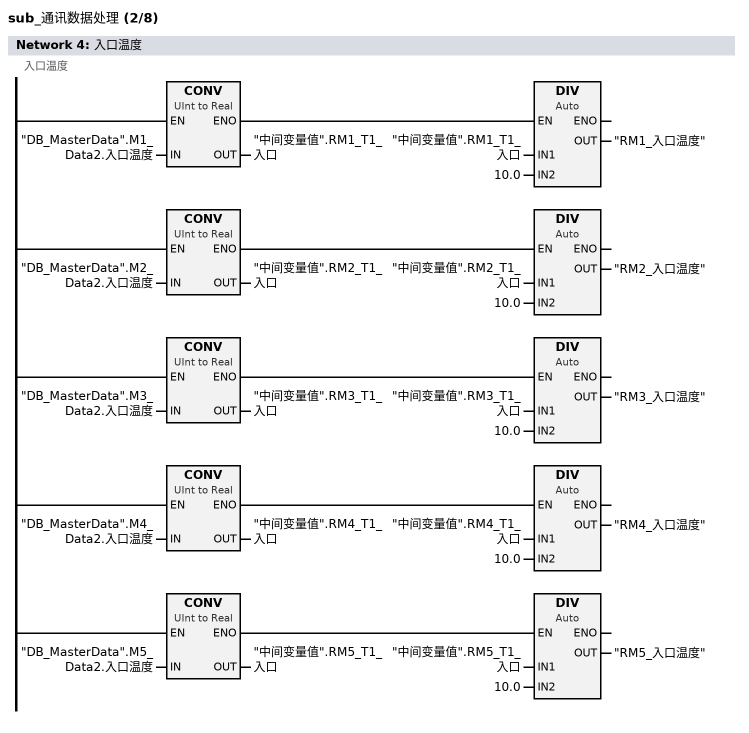
   RUNG wire#powerrail
      { S7_Templates := "[SrcType := UInt, DestType := Real]" } Convert(in := "DB_MasterData".M1_Data2.入口温度, out => "中间变量值".RM1_T1_入口)
      Div(in1 := "中间变量值".RM1_T1_入口, in2 := 10.0, out => "RM1_入口温度")
   END_RUNG
   RUNG wire#powerrail
      { S7_Templates := "[SrcType := UInt, DestType := Real]" } Convert(in := "DB_MasterData".M2_Data2.入口温度, out => "中间变量值".RM2_T1_入口)
      Div(in1 := "中间变量值".RM2_T1_入口, in2 := 10.0, out => "RM2_入口温度")
   END_RUNG
   RUNG wire#powerrail
      { S7_Templates := "[SrcType := UInt, DestType := Real]" } Convert(in := "DB_MasterData".M3_Data2.入口温度, out => "中间变量值".RM3_T1_入口)
      Div(in1 := "中间变量值".RM3_T1_入口, in2 := 10.0, out => "RM3_入口温度")
   END_RUNG
   RUNG wire#powerrail
      { S7_Templates := "[SrcType := UInt, DestType := Real]" } Convert(in := "DB_MasterData".M4_Data2.入口温度, out => "中间变量值".RM4_T1_入口)
      Div(in1 := "中间变量值".RM4_T1_入口, in2 := 10.0, out => "RM4_入口温度")
   END_RUNG
   RUNG wire#powerrail
      { S7_Templates := "[SrcType := UInt, DestType := Real]" } Convert(in := "DB_MasterData".M5_Data2.入口温度, out => "中间变量值".RM5_T1_入口)
      Div(in1 := "中间变量值".RM5_T1_入口, in2 := 10.0, out => "RM5_入口温度")
   END_RUNG
   // the same network as SCL:
   "中间变量值".RM1_T1_入口 := UINT_TO_REAL("DB_MasterData".M1_Data2.入口温度);
   "RM1_入口温度" := "中间变量值".RM1_T1_入口 / 10.0;
   "中间变量值".RM2_T1_入口 := UINT_TO_REAL("DB_MasterData".M2_Data2.入口温度);
   "RM2_入口温度" := "中间变量值".RM2_T1_入口 / 10.0;
   "中间变量值".RM3_T1_入口 := UINT_TO_REAL("DB_MasterData".M3_Data2.入口温度);
   "RM3_入口温度" := "中间变量值".RM3_T1_入口 / 10.0;
   "中间变量值".RM4_T1_入口 := UINT_TO_REAL("DB_MasterData".M4_Data2.入口温度);
   "RM4_入口温度" := "中间变量值".RM4_T1_入口 / 10.0;
   "中间变量值".RM5_T1_入口 := UINT_TO_REAL("DB_MasterData".M5_Data2.入口温度);
   "RM5_入口温度" := "中间变量值".RM5_T1_入口 / 10.0;
END_REGION

REGION Network 5: 出口温度
   // 出口温度
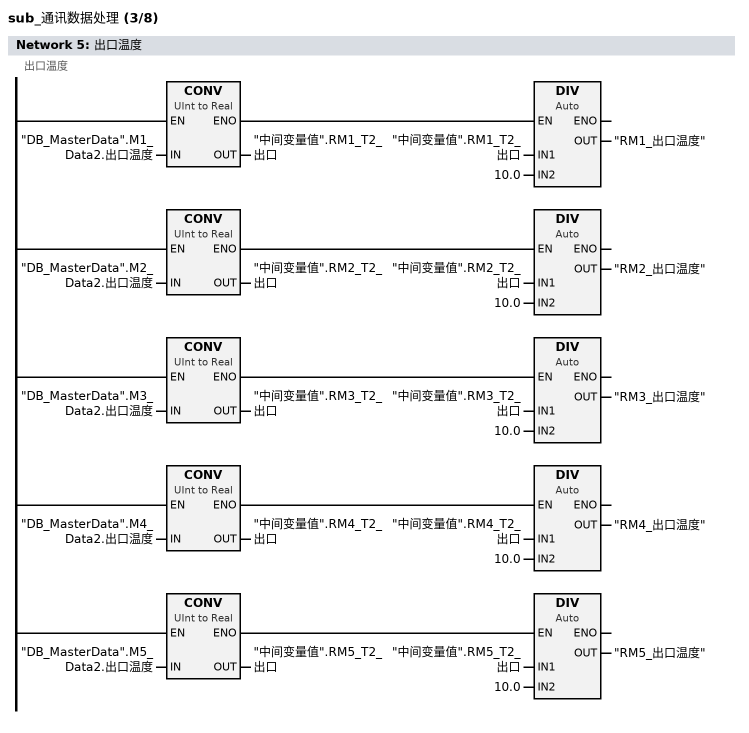
   RUNG wire#powerrail
      { S7_Templates := "[SrcType := UInt, DestType := Real]" } Convert(in := "DB_MasterData".M1_Data2.出口温度, out => "中间变量值".RM1_T2_出口)
      Div(in1 := "中间变量值".RM1_T2_出口, in2 := 10.0, out => "RM1_出口温度")
   END_RUNG
   RUNG wire#powerrail
      { S7_Templates := "[SrcType := UInt, DestType := Real]" } Convert(in := "DB_MasterData".M2_Data2.出口温度, out => "中间变量值".RM2_T2_出口)
      Div(in1 := "中间变量值".RM2_T2_出口, in2 := 10.0, out => "RM2_出口温度")
   END_RUNG
   RUNG wire#powerrail
      { S7_Templates := "[SrcType := UInt, DestType := Real]" } Convert(in := "DB_MasterData".M3_Data2.出口温度, out => "中间变量值".RM3_T2_出口)
      Div(in1 := "中间变量值".RM3_T2_出口, in2 := 10.0, out => "RM3_出口温度")
   END_RUNG
   RUNG wire#powerrail
      { S7_Templates := "[SrcType := UInt, DestType := Real]" } Convert(in := "DB_MasterData".M4_Data2.出口温度, out => "中间变量值".RM4_T2_出口)
      Div(in1 := "中间变量值".RM4_T2_出口, in2 := 10.0, out => "RM4_出口温度")
   END_RUNG
   RUNG wire#powerrail
      { S7_Templates := "[SrcType := UInt, DestType := Real]" } Convert(in := "DB_MasterData".M5_Data2.出口温度, out => "中间变量值".RM5_T2_出口)
      Div(in1 := "中间变量值".RM5_T2_出口, in2 := 10.0, out => "RM5_出口温度")
   END_RUNG
   // the same network as SCL:
   "中间变量值".RM1_T2_出口 := UINT_TO_REAL("DB_MasterData".M1_Data2.出口温度);
   "RM1_出口温度" := "中间变量值".RM1_T2_出口 / 10.0;
   "中间变量值".RM2_T2_出口 := UINT_TO_REAL("DB_MasterData".M2_Data2.出口温度);
   "RM2_出口温度" := "中间变量值".RM2_T2_出口 / 10.0;
   "中间变量值".RM3_T2_出口 := UINT_TO_REAL("DB_MasterData".M3_Data2.出口温度);
   "RM3_出口温度" := "中间变量值".RM3_T2_出口 / 10.0;
   "中间变量值".RM4_T2_出口 := UINT_TO_REAL("DB_MasterData".M4_Data2.出口温度);
   "RM4_出口温度" := "中间变量值".RM4_T2_出口 / 10.0;
   "中间变量值".RM5_T2_出口 := UINT_TO_REAL("DB_MasterData".M5_Data2.出口温度);
   "RM5_出口温度" := "中间变量值".RM5_T2_出口 / 10.0;
END_REGION

REGION Network 7: #1 吸收式热泵数据-温度
   // #1 吸收式热泵数据
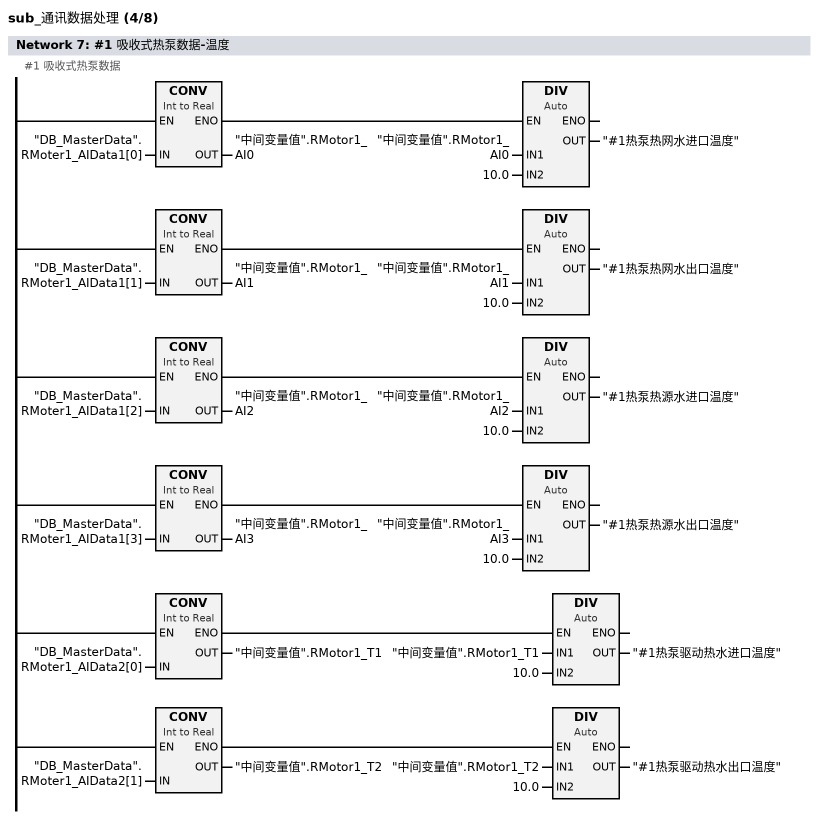
   RUNG wire#powerrail
      { S7_Templates := "[SrcType := Int, DestType := Real]" } Convert(in := "DB_MasterData".RMoter1_AIData1[0], out => "中间变量值".RMotor1_AI0)
      Div(in1 := "中间变量值".RMotor1_AI0, in2 := 10.0, out => "#1热泵热网水进口温度")
   END_RUNG
   RUNG wire#powerrail
      { S7_Templates := "[SrcType := Int, DestType := Real]" } Convert(in := "DB_MasterData".RMoter1_AIData1[1], out => "中间变量值".RMotor1_AI1)
      Div(in1 := "中间变量值".RMotor1_AI1, in2 := 10.0, out => "#1热泵热网水出口温度")
   END_RUNG
   RUNG wire#powerrail
      { S7_Templates := "[SrcType := Int, DestType := Real]" } Convert(in := "DB_MasterData".RMoter1_AIData1[2], out => "中间变量值".RMotor1_AI2)
      Div(in1 := "中间变量值".RMotor1_AI2, in2 := 10.0, out => "#1热泵热源水进口温度")
   END_RUNG
   RUNG wire#powerrail
      { S7_Templates := "[SrcType := Int, DestType := Real]" } Convert(in := "DB_MasterData".RMoter1_AIData1[3], out => "中间变量值".RMotor1_AI3)
      Div(in1 := "中间变量值".RMotor1_AI3, in2 := 10.0, out => "#1热泵热源水出口温度")
   END_RUNG
   RUNG wire#powerrail
      { S7_Templates := "[SrcType := Int, DestType := Real]" } Convert(in := "DB_MasterData".RMoter1_AIData2[0], out => "中间变量值".RMotor1_T1)
      Div(in1 := "中间变量值".RMotor1_T1, in2 := 10.0, out => "#1热泵驱动热水进口温度")
   END_RUNG
   RUNG wire#powerrail
      { S7_Templates := "[SrcType := Int, DestType := Real]" } Convert(in := "DB_MasterData".RMoter1_AIData2[1], out => "中间变量值".RMotor1_T2)
      Div(in1 := "中间变量值".RMotor1_T2, in2 := 10.0, out => "#1热泵驱动热水出口温度")
   END_RUNG
   // the same network as SCL:
   "中间变量值".RMotor1_AI0 := INT_TO_REAL("DB_MasterData".RMoter1_AIData1[0]);
   "#1热泵热网水进口温度" := "中间变量值".RMotor1_AI0 / 10.0;
   "中间变量值".RMotor1_AI1 := INT_TO_REAL("DB_MasterData".RMoter1_AIData1[1]);
   "#1热泵热网水出口温度" := "中间变量值".RMotor1_AI1 / 10.0;
   "中间变量值".RMotor1_AI2 := INT_TO_REAL("DB_MasterData".RMoter1_AIData1[2]);
   "#1热泵热源水进口温度" := "中间变量值".RMotor1_AI2 / 10.0;
   "中间变量值".RMotor1_AI3 := INT_TO_REAL("DB_MasterData".RMoter1_AIData1[3]);
   "#1热泵热源水出口温度" := "中间变量值".RMotor1_AI3 / 10.0;
   "中间变量值".RMotor1_T1 := INT_TO_REAL("DB_MasterData".RMoter1_AIData2[0]);
   "#1热泵驱动热水进口温度" := "中间变量值".RMotor1_T1 / 10.0;
   "中间变量值".RMotor1_T2 := INT_TO_REAL("DB_MasterData".RMoter1_AIData2[1]);
   "#1热泵驱动热水出口温度" := "中间变量值".RMotor1_T2 / 10.0;
END_REGION

REGION Network 8: #1 吸收式热泵数据-压力
   // #1 吸收式热泵数据-压力
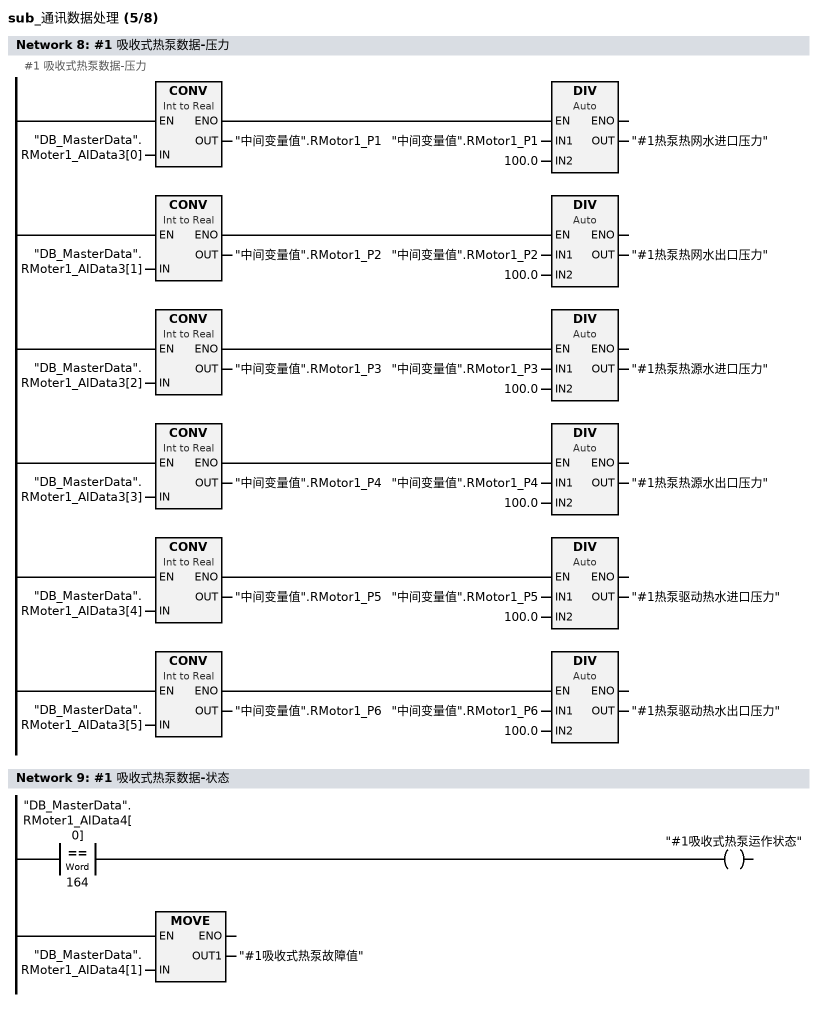
   RUNG wire#powerrail
      { S7_Templates := "[SrcType := Int, DestType := Real]" } Convert(in := "DB_MasterData".RMoter1_AIData3[0], out => "中间变量值".RMotor1_P1)
      Div(in1 := "中间变量值".RMotor1_P1, in2 := 100.0, out => "#1热泵热网水进口压力")
   END_RUNG
   RUNG wire#powerrail
      { S7_Templates := "[SrcType := Int, DestType := Real]" } Convert(in := "DB_MasterData".RMoter1_AIData3[1], out => "中间变量值".RMotor1_P2)
      Div(in1 := "中间变量值".RMotor1_P2, in2 := 100.0, out => "#1热泵热网水出口压力")
   END_RUNG
   RUNG wire#powerrail
      { S7_Templates := "[SrcType := Int, DestType := Real]" } Convert(in := "DB_MasterData".RMoter1_AIData3[2], out => "中间变量值".RMotor1_P3)
      Div(in1 := "中间变量值".RMotor1_P3, in2 := 100.0, out => "#1热泵热源水进口压力")
   END_RUNG
   RUNG wire#powerrail
      { S7_Templates := "[SrcType := Int, DestType := Real]" } Convert(in := "DB_MasterData".RMoter1_AIData3[3], out => "中间变量值".RMotor1_P4)
      Div(in1 := "中间变量值".RMotor1_P4, in2 := 100.0, out => "#1热泵热源水出口压力")
   END_RUNG
   RUNG wire#powerrail
      { S7_Templates := "[SrcType := Int, DestType := Real]" } Convert(in := "DB_MasterData".RMoter1_AIData3[4], out => "中间变量值".RMotor1_P5)
      Div(in1 := "中间变量值".RMotor1_P5, in2 := 100.0, out => "#1热泵驱动热水进口压力")
   END_RUNG
   RUNG wire#powerrail
      { S7_Templates := "[SrcType := Int, DestType := Real]" } Convert(in := "DB_MasterData".RMoter1_AIData3[5], out => "中间变量值".RMotor1_P6)
      Div(in1 := "中间变量值".RMotor1_P6, in2 := 100.0, out => "#1热泵驱动热水出口压力")
   END_RUNG
   // the same network as SCL:
   "中间变量值".RMotor1_P1 := INT_TO_REAL("DB_MasterData".RMoter1_AIData3[0]);
   "#1热泵热网水进口压力" := "中间变量值".RMotor1_P1 / 100.0;
   "中间变量值".RMotor1_P2 := INT_TO_REAL("DB_MasterData".RMoter1_AIData3[1]);
   "#1热泵热网水出口压力" := "中间变量值".RMotor1_P2 / 100.0;
   "中间变量值".RMotor1_P3 := INT_TO_REAL("DB_MasterData".RMoter1_AIData3[2]);
   "#1热泵热源水进口压力" := "中间变量值".RMotor1_P3 / 100.0;
   "中间变量值".RMotor1_P4 := INT_TO_REAL("DB_MasterData".RMoter1_AIData3[3]);
   "#1热泵热源水出口压力" := "中间变量值".RMotor1_P4 / 100.0;
   "中间变量值".RMotor1_P5 := INT_TO_REAL("DB_MasterData".RMoter1_AIData3[4]);
   "#1热泵驱动热水进口压力" := "中间变量值".RMotor1_P5 / 100.0;
   "中间变量值".RMotor1_P6 := INT_TO_REAL("DB_MasterData".RMoter1_AIData3[5]);
   "#1热泵驱动热水出口压力" := "中间变量值".RMotor1_P6 / 100.0;
END_REGION

REGION Network 9: #1 吸收式热泵数据-状态
   RUNG wire#powerrail
      { S7_Templates := "SrcType := Word" } EQ_Contact(in1 := "DB_MasterData".RMoter1_AIData4[0], in2 := 164)
      Coil( "#1吸收式热泵运作状态" )
   END_RUNG
   RUNG wire#powerrail
      Move(in := "DB_MasterData".RMoter1_AIData4[1], out1 => "#1吸收式热泵故障值")
   END_RUNG
   // the same network as SCL:
   "#1吸收式热泵运作状态" := "DB_MasterData".RMoter1_AIData4[0] = 164;
   "#1吸收式热泵故障值" := "DB_MasterData".RMoter1_AIData4[1];
END_REGION

REGION Network 10: #2 吸收式热泵数据-温度
   // #2 吸收式热泵数据
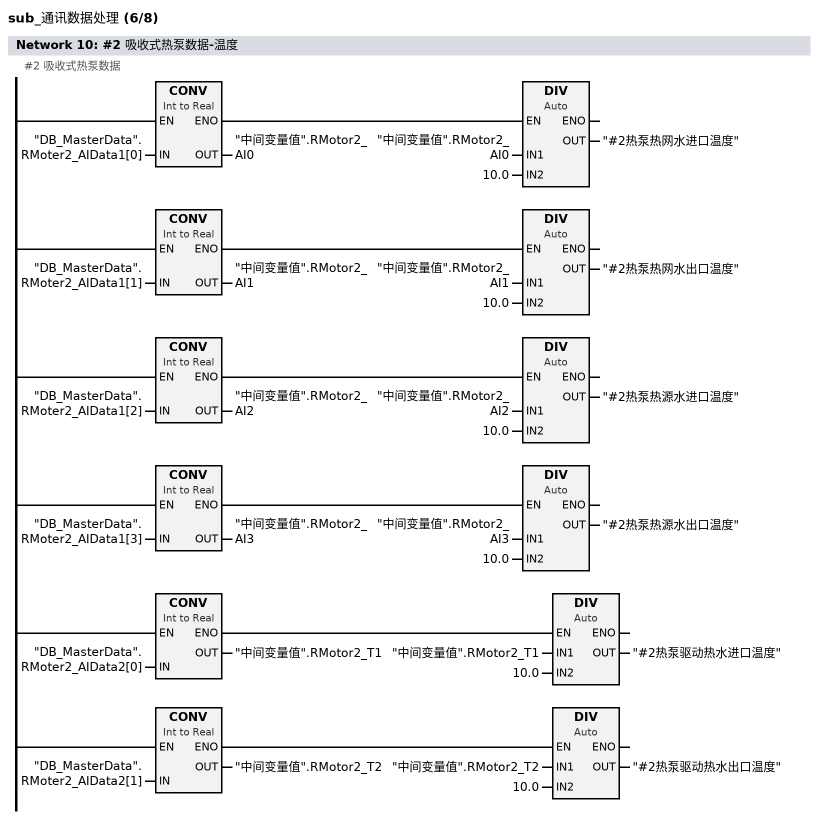
   RUNG wire#powerrail
      { S7_Templates := "[SrcType := Int, DestType := Real]" } Convert(in := "DB_MasterData".RMoter2_AIData1[0], out => "中间变量值".RMotor2_AI0)
      Div(in1 := "中间变量值".RMotor2_AI0, in2 := 10.0, out => "#2热泵热网水进口温度")
   END_RUNG
   RUNG wire#powerrail
      { S7_Templates := "[SrcType := Int, DestType := Real]" } Convert(in := "DB_MasterData".RMoter2_AIData1[1], out => "中间变量值".RMotor2_AI1)
      Div(in1 := "中间变量值".RMotor2_AI1, in2 := 10.0, out => "#2热泵热网水出口温度")
   END_RUNG
   RUNG wire#powerrail
      { S7_Templates := "[SrcType := Int, DestType := Real]" } Convert(in := "DB_MasterData".RMoter2_AIData1[2], out => "中间变量值".RMotor2_AI2)
      Div(in1 := "中间变量值".RMotor2_AI2, in2 := 10.0, out => "#2热泵热源水进口温度")
   END_RUNG
   RUNG wire#powerrail
      { S7_Templates := "[SrcType := Int, DestType := Real]" } Convert(in := "DB_MasterData".RMoter2_AIData1[3], out => "中间变量值".RMotor2_AI3)
      Div(in1 := "中间变量值".RMotor2_AI3, in2 := 10.0, out => "#2热泵热源水出口温度")
   END_RUNG
   RUNG wire#powerrail
      { S7_Templates := "[SrcType := Int, DestType := Real]" } Convert(in := "DB_MasterData".RMoter2_AIData2[0], out => "中间变量值".RMotor2_T1)
      Div(in1 := "中间变量值".RMotor2_T1, in2 := 10.0, out => "#2热泵驱动热水进口温度")
   END_RUNG
   RUNG wire#powerrail
      { S7_Templates := "[SrcType := Int, DestType := Real]" } Convert(in := "DB_MasterData".RMoter2_AIData2[1], out => "中间变量值".RMotor2_T2)
      Div(in1 := "中间变量值".RMotor2_T2, in2 := 10.0, out => "#2热泵驱动热水出口温度")
   END_RUNG
   // the same network as SCL:
   "中间变量值".RMotor2_AI0 := INT_TO_REAL("DB_MasterData".RMoter2_AIData1[0]);
   "#2热泵热网水进口温度" := "中间变量值".RMotor2_AI0 / 10.0;
   "中间变量值".RMotor2_AI1 := INT_TO_REAL("DB_MasterData".RMoter2_AIData1[1]);
   "#2热泵热网水出口温度" := "中间变量值".RMotor2_AI1 / 10.0;
   "中间变量值".RMotor2_AI2 := INT_TO_REAL("DB_MasterData".RMoter2_AIData1[2]);
   "#2热泵热源水进口温度" := "中间变量值".RMotor2_AI2 / 10.0;
   "中间变量值".RMotor2_AI3 := INT_TO_REAL("DB_MasterData".RMoter2_AIData1[3]);
   "#2热泵热源水出口温度" := "中间变量值".RMotor2_AI3 / 10.0;
   "中间变量值".RMotor2_T1 := INT_TO_REAL("DB_MasterData".RMoter2_AIData2[0]);
   "#2热泵驱动热水进口温度" := "中间变量值".RMotor2_T1 / 10.0;
   "中间变量值".RMotor2_T2 := INT_TO_REAL("DB_MasterData".RMoter2_AIData2[1]);
   "#2热泵驱动热水出口温度" := "中间变量值".RMotor2_T2 / 10.0;
END_REGION

REGION Network 11: #2吸收式热泵数据-压力
   // #2 吸收式热泵数据-压力
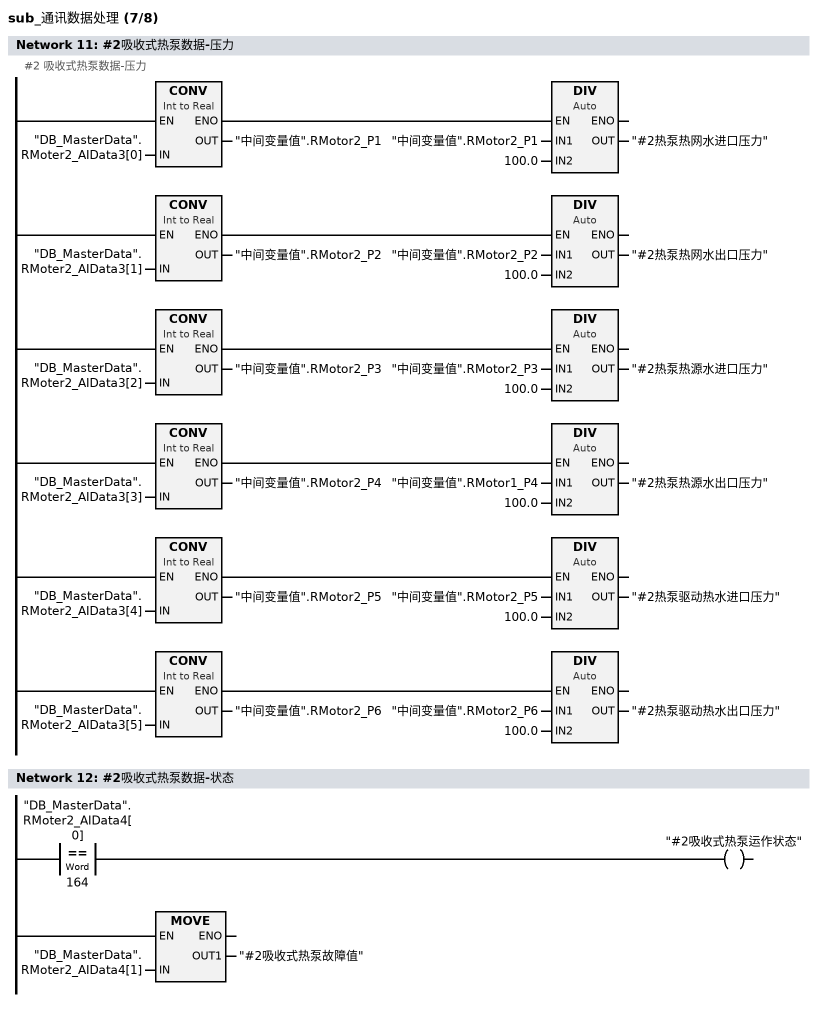
   RUNG wire#powerrail
      { S7_Templates := "[SrcType := Int, DestType := Real]" } Convert(in := "DB_MasterData".RMoter2_AIData3[0], out => "中间变量值".RMotor2_P1)
      Div(in1 := "中间变量值".RMotor2_P1, in2 := 100.0, out => "#2热泵热网水进口压力")
   END_RUNG
   RUNG wire#powerrail
      { S7_Templates := "[SrcType := Int, DestType := Real]" } Convert(in := "DB_MasterData".RMoter2_AIData3[1], out => "中间变量值".RMotor2_P2)
      Div(in1 := "中间变量值".RMotor2_P2, in2 := 100.0, out => "#2热泵热网水出口压力")
   END_RUNG
   RUNG wire#powerrail
      { S7_Templates := "[SrcType := Int, DestType := Real]" } Convert(in := "DB_MasterData".RMoter2_AIData3[2], out => "中间变量值".RMotor2_P3)
      Div(in1 := "中间变量值".RMotor2_P3, in2 := 100.0, out => "#2热泵热源水进口压力")
   END_RUNG
   RUNG wire#powerrail
      { S7_Templates := "[SrcType := Int, DestType := Real]" } Convert(in := "DB_MasterData".RMoter2_AIData3[3], out => "中间变量值".RMotor2_P4)
      Div(in1 := "中间变量值".RMotor1_P4, in2 := 100.0, out => "#2热泵热源水出口压力")
   END_RUNG
   RUNG wire#powerrail
      { S7_Templates := "[SrcType := Int, DestType := Real]" } Convert(in := "DB_MasterData".RMoter2_AIData3[4], out => "中间变量值".RMotor2_P5)
      Div(in1 := "中间变量值".RMotor2_P5, in2 := 100.0, out => "#2热泵驱动热水进口压力")
   END_RUNG
   RUNG wire#powerrail
      { S7_Templates := "[SrcType := Int, DestType := Real]" } Convert(in := "DB_MasterData".RMoter2_AIData3[5], out => "中间变量值".RMotor2_P6)
      Div(in1 := "中间变量值".RMotor2_P6, in2 := 100.0, out => "#2热泵驱动热水出口压力")
   END_RUNG
   // the same network as SCL:
   "中间变量值".RMotor2_P1 := INT_TO_REAL("DB_MasterData".RMoter2_AIData3[0]);
   "#2热泵热网水进口压力" := "中间变量值".RMotor2_P1 / 100.0;
   "中间变量值".RMotor2_P2 := INT_TO_REAL("DB_MasterData".RMoter2_AIData3[1]);
   "#2热泵热网水出口压力" := "中间变量值".RMotor2_P2 / 100.0;
   "中间变量值".RMotor2_P3 := INT_TO_REAL("DB_MasterData".RMoter2_AIData3[2]);
   "#2热泵热源水进口压力" := "中间变量值".RMotor2_P3 / 100.0;
   "中间变量值".RMotor2_P4 := INT_TO_REAL("DB_MasterData".RMoter2_AIData3[3]);
   "#2热泵热源水出口压力" := "中间变量值".RMotor1_P4 / 100.0;
   "中间变量值".RMotor2_P5 := INT_TO_REAL("DB_MasterData".RMoter2_AIData3[4]);
   "#2热泵驱动热水进口压力" := "中间变量值".RMotor2_P5 / 100.0;
   "中间变量值".RMotor2_P6 := INT_TO_REAL("DB_MasterData".RMoter2_AIData3[5]);
   "#2热泵驱动热水出口压力" := "中间变量值".RMotor2_P6 / 100.0;
END_REGION

REGION Network 12: #2吸收式热泵数据-状态
   RUNG wire#powerrail
      { S7_Templates := "SrcType := Word" } EQ_Contact(in1 := "DB_MasterData".RMoter2_AIData4[0], in2 := 164)
      Coil( "#2吸收式热泵运作状态" )
   END_RUNG
   RUNG wire#powerrail
      Move(in := "DB_MasterData".RMoter2_AIData4[1], out1 => "#2吸收式热泵故障值")
   END_RUNG
   // the same network as SCL:
   "#2吸收式热泵运作状态" := "DB_MasterData".RMoter2_AIData4[0] = 164;
   "#2吸收式热泵故障值" := "DB_MasterData".RMoter2_AIData4[1];
END_REGION

REGION Network 14
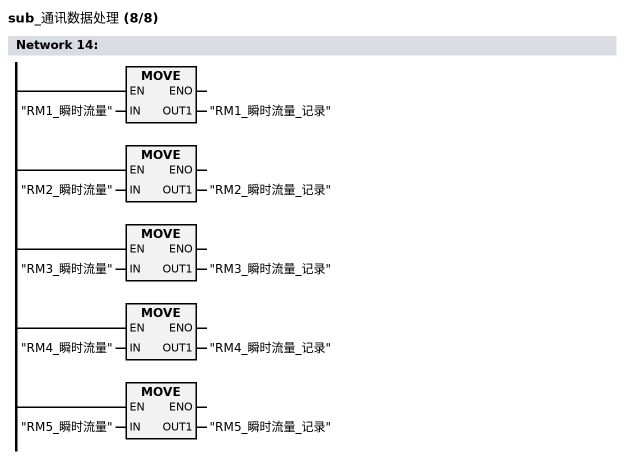
   RUNG wire#powerrail
      Move(in := "RM1_瞬时流量", out1 => "RM1_瞬时流量_记录")
   END_RUNG
   RUNG wire#powerrail
      Move(in := "RM2_瞬时流量", out1 => "RM2_瞬时流量_记录")
   END_RUNG
   RUNG wire#powerrail
      Move(in := "RM3_瞬时流量", out1 => "RM3_瞬时流量_记录")
   END_RUNG
   RUNG wire#powerrail
      Move(in := "RM4_瞬时流量", out1 => "RM4_瞬时流量_记录")
   END_RUNG
   RUNG wire#powerrail
      Move(in := "RM5_瞬时流量", out1 => "RM5_瞬时流量_记录")
   END_RUNG
   // the same network as SCL:
   "RM1_瞬时流量_记录" := "RM1_瞬时流量";
   "RM2_瞬时流量_记录" := "RM2_瞬时流量";
   "RM3_瞬时流量_记录" := "RM3_瞬时流量";
   "RM4_瞬时流量_记录" := "RM4_瞬时流量";
   "RM5_瞬时流量_记录" := "RM5_瞬时流量";
END_REGION
END_ORGANIZATION_BLOCK

ORGANIZATION_BLOCK "sub_自动逻辑"   // OB125, LAD, ProgramCycle
TITLE = "Main Program Sweep (Cycle)"
{ S7_Optimized_Access := 'TRUE' }
VERSION : 0.1
   VAR_INPUT
      Initial_Call : Bool;   // Initial call of this OB
      Remanence : Bool;   // =True, if remanent data are available
   END_VAR
   VAR_TEMP   // added for the SCL form of the ladder/FBD networks
      _w1 : Bool;
      _w2 : Bool;
      _w3 : Bool;
      _w4 : Bool;
      _w5 : Bool;
      _w6 : Bool;
      _w7 : Bool;
      _w8 : Bool;
   END_VAR
BEGIN

REGION Network 1: 自动补水逻辑-停止逻辑
   // 补水泵停止逻辑
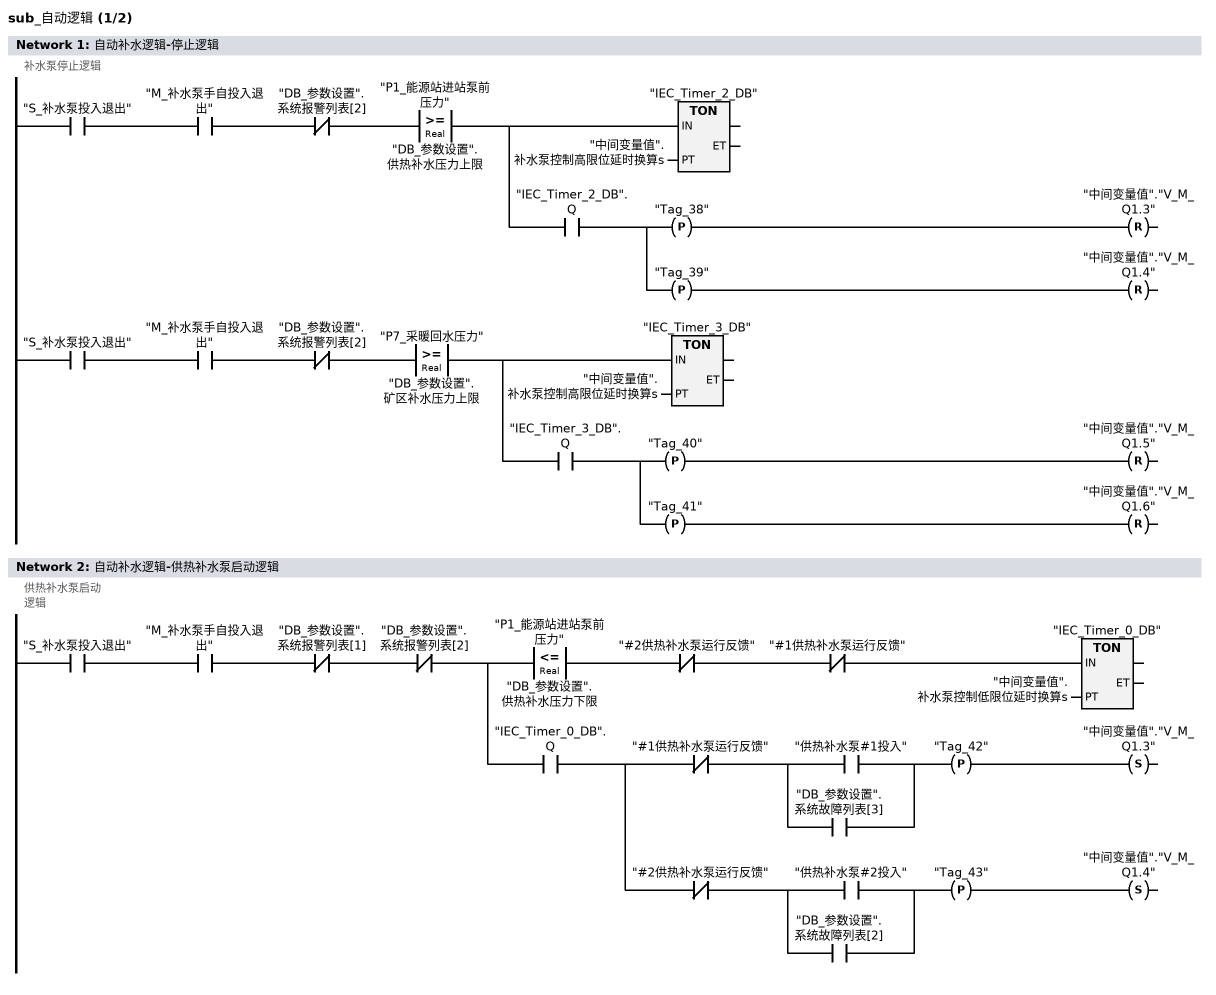
   #_w1 := "S_补水泵投入退出" AND "M_补水泵手自投入退出" AND NOT "DB_参数设置".系统报警列表[2] AND ("P1_能源站进站泵前压力" >= "DB_参数设置".供热补水压力上限);
   "IEC_Timer_2_DB".TON(IN := #_w1, PT := "中间变量值".补水泵控制高限位延时换算s);
   #_w2 := #_w1 AND "IEC_Timer_2_DB".Q;
   #_w3 := #_w2 AND NOT "Tag_38";   // rising edge
   "Tag_38" := #_w2;
   IF #_w3 THEN "中间变量值"."V_M_Q1.3" := FALSE; END_IF;
   #_w4 := #_w2 AND NOT "Tag_39";   // rising edge
   "Tag_39" := #_w2;
   IF #_w4 THEN "中间变量值"."V_M_Q1.4" := FALSE; END_IF;
   #_w5 := "S_补水泵投入退出" AND "M_补水泵手自投入退出" AND NOT "DB_参数设置".系统报警列表[2] AND ("P7_采暖回水压力" >= "DB_参数设置".矿区补水压力上限);
   "IEC_Timer_3_DB".TON(IN := #_w5, PT := "中间变量值".补水泵控制高限位延时换算s);
   #_w6 := #_w5 AND "IEC_Timer_3_DB".Q;
   #_w7 := #_w6 AND NOT "Tag_40";   // rising edge
   "Tag_40" := #_w6;
   IF #_w7 THEN "中间变量值"."V_M_Q1.5" := FALSE; END_IF;
   #_w8 := #_w6 AND NOT "Tag_41";   // rising edge
   "Tag_41" := #_w6;
   IF #_w8 THEN "中间变量值"."V_M_Q1.6" := FALSE; END_IF;
END_REGION

REGION Network 2: 自动补水逻辑-供热补水泵启动逻辑
   // 供热补水泵启动
   // 逻辑
   #_w1 := "S_补水泵投入退出" AND "M_补水泵手自投入退出" AND NOT "DB_参数设置".系统报警列表[1] AND NOT "DB_参数设置".系统报警列表[2];
   "IEC_Timer_0_DB".TON(IN := #_w1 AND ("P1_能源站进站泵前压力" <= "DB_参数设置".供热补水压力下限) AND NOT "#2供热补水泵运行反馈" AND NOT "#1供热补水泵运行反馈",
                        PT := "中间变量值".补水泵控制低限位延时换算s);
   #_w2 := #_w1 AND "IEC_Timer_0_DB".Q;
   #_w3 := #_w2 AND NOT "#1供热补水泵运行反馈" AND ("供热补水泵#1投入" OR "DB_参数设置".系统故障列表[3]);
   #_w4 := #_w3 AND NOT "Tag_42";   // rising edge
   "Tag_42" := #_w3;
   IF #_w4 THEN "中间变量值"."V_M_Q1.3" := TRUE; END_IF;
   #_w5 := #_w2 AND NOT "#2供热补水泵运行反馈" AND ("供热补水泵#2投入" OR "DB_参数设置".系统故障列表[2]);
   #_w6 := #_w5 AND NOT "Tag_43";   // rising edge
   "Tag_43" := #_w5;
   IF #_w6 THEN "中间变量值"."V_M_Q1.4" := TRUE; END_IF;
END_REGION

REGION Network 3: 自动补水逻辑 矿区补水泵启动逻辑
   // 矿区补水泵启动逻辑
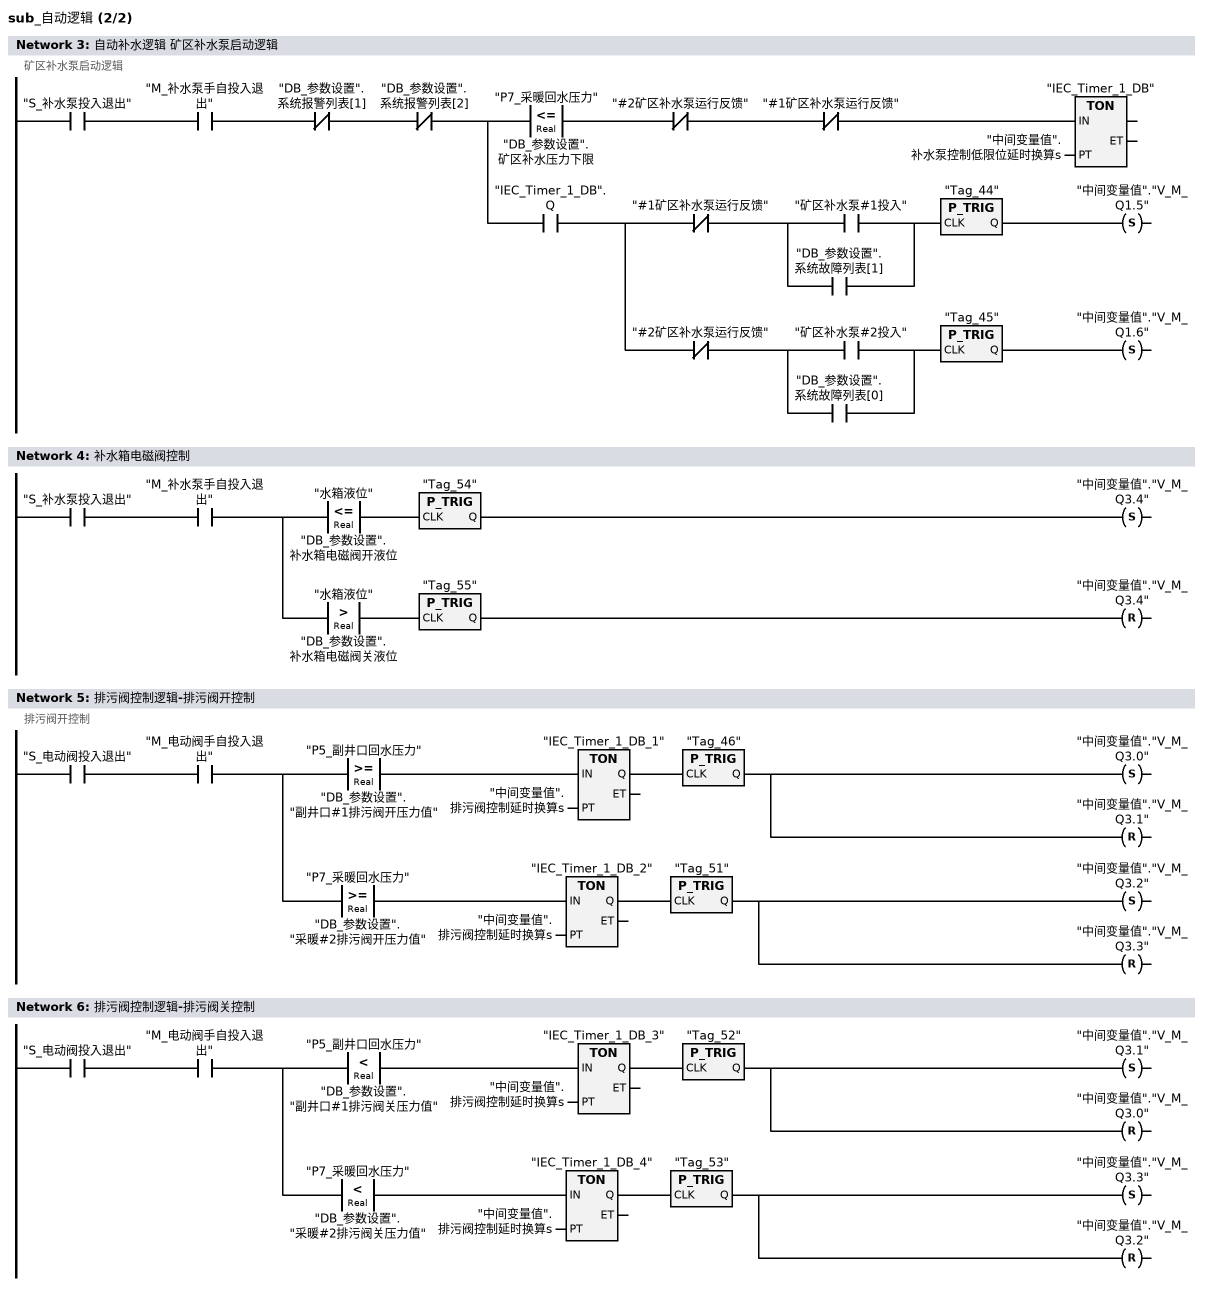
   #_w1 := "S_补水泵投入退出" AND "M_补水泵手自投入退出" AND NOT "DB_参数设置".系统报警列表[1] AND NOT "DB_参数设置".系统报警列表[2];
   "IEC_Timer_1_DB".TON(IN := #_w1 AND ("P7_采暖回水压力" <= "DB_参数设置".矿区补水压力下限) AND NOT "#2矿区补水泵运行反馈" AND NOT "#1矿区补水泵运行反馈",
                        PT := "中间变量值".补水泵控制低限位延时换算s);
   #_w2 := #_w1 AND "IEC_Timer_1_DB".Q;
   #_w3 := #_w2 AND NOT "#1矿区补水泵运行反馈" AND ("矿区补水泵#1投入" OR "DB_参数设置".系统故障列表[1]);
   #_w4 := #_w3 AND NOT "Tag_44";   // rising edge
   "Tag_44" := #_w3;
   IF #_w4 THEN "中间变量值"."V_M_Q1.5" := TRUE; END_IF;
   #_w5 := #_w2 AND NOT "#2矿区补水泵运行反馈" AND ("矿区补水泵#2投入" OR "DB_参数设置".系统故障列表[0]);
   #_w6 := #_w5 AND NOT "Tag_45";   // rising edge
   "Tag_45" := #_w5;
   IF #_w6 THEN "中间变量值"."V_M_Q1.6" := TRUE; END_IF;
END_REGION

REGION Network 4: 补水箱电磁阀控制
   RUNG wire#powerrail
      Contact( "S_补水泵投入退出" )
      Contact( "M_补水泵手自投入退出" )
      wire#w1
      { S7_Templates := "SrcType := Real" } LE_Contact(in1 := "水箱液位", in2 := "DB_参数设置".补水箱电磁阀开液位)
      P_Trig( "Tag_54" )
      S_Coil( "中间变量值"."V_M_Q3.4" )
   END_RUNG
   RUNG wire#w1
      { S7_Templates := "SrcType := Real" } GT_Contact(in1 := "水箱液位", in2 := "DB_参数设置".补水箱电磁阀关液位)
      P_Trig( "Tag_55" )
      R_Coil( "中间变量值"."V_M_Q3.4" )
   END_RUNG
   // the same network as SCL:
   #_w1 := "S_补水泵投入退出" AND "M_补水泵手自投入退出";
   #_w2 := #_w1 AND ("水箱液位" <= "DB_参数设置".补水箱电磁阀开液位);
   #_w3 := #_w2 AND NOT "Tag_54";   // rising edge
   "Tag_54" := #_w2;
   IF #_w3 THEN "中间变量值"."V_M_Q3.4" := TRUE; END_IF;
   #_w4 := #_w1 AND ("水箱液位" > "DB_参数设置".补水箱电磁阀关液位);
   #_w5 := #_w4 AND NOT "Tag_55";   // rising edge
   "Tag_55" := #_w4;
   IF #_w5 THEN "中间变量值"."V_M_Q3.4" := FALSE; END_IF;
END_REGION

REGION Network 5: 排污阀控制逻辑-排污阀开控制
   // 排污阀开控制
   #_w1 := "S_电动阀投入退出" AND "M_电动阀手自投入退出";
   "IEC_Timer_1_DB_1".TON(IN := #_w1 AND ("P5_副井口回水压力" >= "DB_参数设置"."副井口#1排污阀开压力值"), PT := "中间变量值".排污阀控制延时换算s);
   #_w2 := "IEC_Timer_1_DB_1".Q AND NOT "Tag_46";   // rising edge
   "Tag_46" := "IEC_Timer_1_DB_1".Q;
   IF #_w2 THEN
       "中间变量值"."V_M_Q3.0" := TRUE;
       "中间变量值"."V_M_Q3.1" := FALSE;
   END_IF;
   "IEC_Timer_1_DB_2".TON(IN := #_w1 AND ("P7_采暖回水压力" >= "DB_参数设置"."采暖#2排污阀开压力值"), PT := "中间变量值".排污阀控制延时换算s);
   #_w3 := "IEC_Timer_1_DB_2".Q AND NOT "Tag_51";   // rising edge
   "Tag_51" := "IEC_Timer_1_DB_2".Q;
   IF #_w3 THEN
       "中间变量值"."V_M_Q3.2" := TRUE;
       "中间变量值"."V_M_Q3.3" := FALSE;
   END_IF;
END_REGION

REGION Network 6: 排污阀控制逻辑-排污阀关控制
   #_w1 := "S_电动阀投入退出" AND "M_电动阀手自投入退出";
   "IEC_Timer_1_DB_3".TON(IN := #_w1 AND ("P5_副井口回水压力" < "DB_参数设置"."副井口#1排污阀关压力值"), PT := "中间变量值".排污阀控制延时换算s);
   #_w2 := "IEC_Timer_1_DB_3".Q AND NOT "Tag_52";   // rising edge
   "Tag_52" := "IEC_Timer_1_DB_3".Q;
   IF #_w2 THEN
       "中间变量值"."V_M_Q3.1" := TRUE;
       "中间变量值"."V_M_Q3.0" := FALSE;
   END_IF;
   "IEC_Timer_1_DB_4".TON(IN := #_w1 AND ("P7_采暖回水压力" < "DB_参数设置"."采暖#2排污阀关压力值"), PT := "中间变量值".排污阀控制延时换算s);
   #_w3 := "IEC_Timer_1_DB_4".Q AND NOT "Tag_53";   // rising edge
   "Tag_53" := "IEC_Timer_1_DB_4".Q;
   IF #_w3 THEN
       "中间变量值"."V_M_Q3.3" := TRUE;
       "中间变量值"."V_M_Q3.2" := FALSE;
   END_IF;
END_REGION
END_ORGANIZATION_BLOCK

ORGANIZATION_BLOCK "sub_手动操作"   // OB126, LAD, ProgramCycle
TITLE = "Main Program Sweep (Cycle)"
{ S7_Optimized_Access := 'TRUE' }
VERSION : 0.1
   VAR_INPUT
      Initial_Call : Bool;   // Initial call of this OB
      Remanence : Bool;   // =True, if remanent data are available
   END_VAR
   VAR_TEMP   // added for the SCL form of the ladder/FBD networks
      _w1 : Bool;
      _w2 : Bool;
      _w3 : Bool;
      _w4 : Bool;
      _w5 : Bool;
      _w6 : Bool;
   END_VAR
BEGIN

REGION Network 1: #1隔离泵控制输出中间变量
   // #1采暖泵
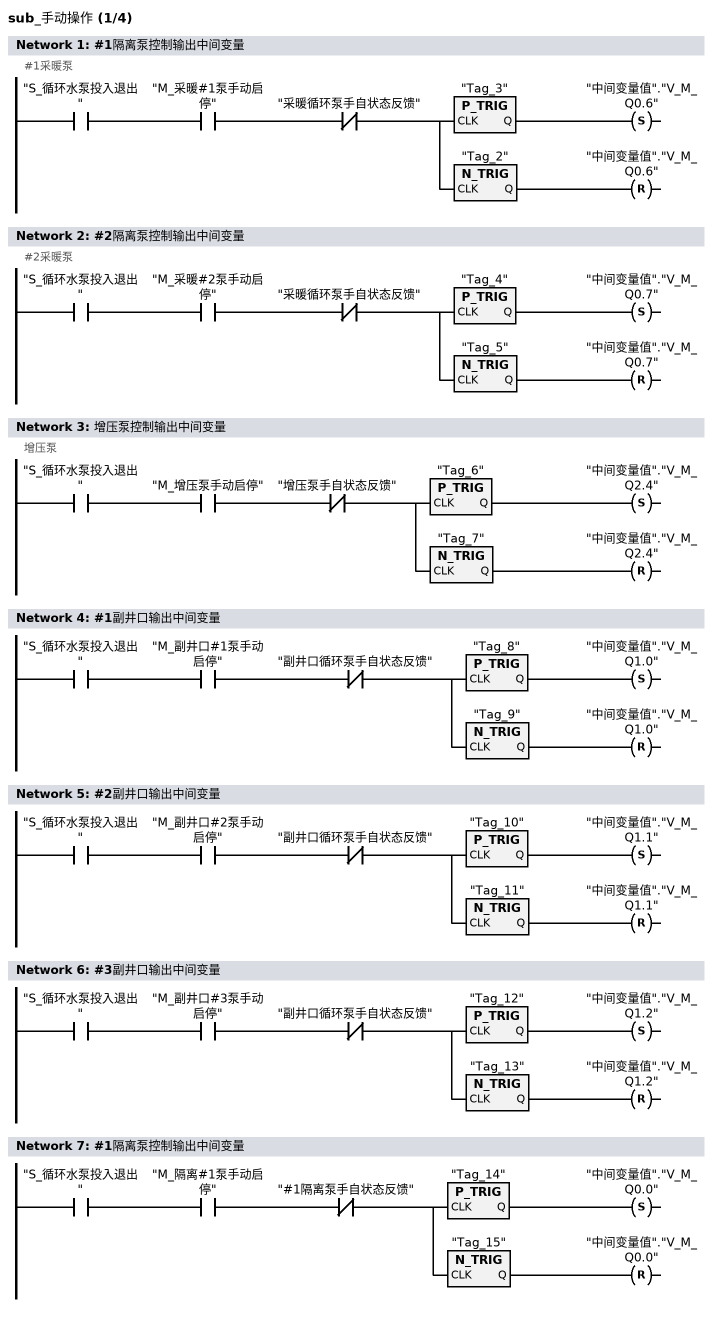
   RUNG wire#powerrail
      Contact( "S_循环水泵投入退出" )
      Contact( "M_采暖#1泵手动启停" )
      I_Contact( "采暖循环泵手自状态反馈" )
      wire#w1
      P_Trig( "Tag_3" )
      S_Coil( "中间变量值"."V_M_Q0.6" )
   END_RUNG
   RUNG wire#w1
      N_Trig( "Tag_2" )
      R_Coil( "中间变量值"."V_M_Q0.6" )
   END_RUNG
   // the same network as SCL:
   #_w1 := "S_循环水泵投入退出" AND "M_采暖#1泵手动启停" AND NOT "采暖循环泵手自状态反馈";
   #_w2 := #_w1 AND NOT "Tag_3";   // rising edge
   "Tag_3" := #_w1;
   IF #_w2 THEN "中间变量值"."V_M_Q0.6" := TRUE; END_IF;
   #_w3 := NOT #_w1 AND "Tag_2";   // falling edge
   "Tag_2" := #_w1;
   IF #_w3 THEN "中间变量值"."V_M_Q0.6" := FALSE; END_IF;
END_REGION

REGION Network 2: #2隔离泵控制输出中间变量
   // #2采暖泵
   RUNG wire#powerrail
      Contact( "S_循环水泵投入退出" )
      Contact( "M_采暖#2泵手动启停" )
      I_Contact( "采暖循环泵手自状态反馈" )
      wire#w1
      P_Trig( "Tag_4" )
      S_Coil( "中间变量值"."V_M_Q0.7" )
   END_RUNG
   RUNG wire#w1
      N_Trig( "Tag_5" )
      R_Coil( "中间变量值"."V_M_Q0.7" )
   END_RUNG
   // the same network as SCL:
   #_w1 := "S_循环水泵投入退出" AND "M_采暖#2泵手动启停" AND NOT "采暖循环泵手自状态反馈";
   #_w2 := #_w1 AND NOT "Tag_4";   // rising edge
   "Tag_4" := #_w1;
   IF #_w2 THEN "中间变量值"."V_M_Q0.7" := TRUE; END_IF;
   #_w3 := NOT #_w1 AND "Tag_5";   // falling edge
   "Tag_5" := #_w1;
   IF #_w3 THEN "中间变量值"."V_M_Q0.7" := FALSE; END_IF;
END_REGION

REGION Network 3: 增压泵控制输出中间变量
   // 增压泵
   RUNG wire#powerrail
      Contact( "S_循环水泵投入退出" )
      Contact( "M_增压泵手动启停" )
      I_Contact( "增压泵手自状态反馈" )
      wire#w1
      P_Trig( "Tag_6" )
      S_Coil( "中间变量值"."V_M_Q2.4" )
   END_RUNG
   RUNG wire#w1
      N_Trig( "Tag_7" )
      R_Coil( "中间变量值"."V_M_Q2.4" )
   END_RUNG
   // the same network as SCL:
   #_w1 := "S_循环水泵投入退出" AND "M_增压泵手动启停" AND NOT "增压泵手自状态反馈";
   #_w2 := #_w1 AND NOT "Tag_6";   // rising edge
   "Tag_6" := #_w1;
   IF #_w2 THEN "中间变量值"."V_M_Q2.4" := TRUE; END_IF;
   #_w3 := NOT #_w1 AND "Tag_7";   // falling edge
   "Tag_7" := #_w1;
   IF #_w3 THEN "中间变量值"."V_M_Q2.4" := FALSE; END_IF;
END_REGION

REGION Network 4: #1副井口输出中间变量
   RUNG wire#powerrail
      Contact( "S_循环水泵投入退出" )
      Contact( "M_副井口#1泵手动启停" )
      I_Contact( "副井口循环泵手自状态反馈" )
      wire#w1
      P_Trig( "Tag_8" )
      S_Coil( "中间变量值"."V_M_Q1.0" )
   END_RUNG
   RUNG wire#w1
      N_Trig( "Tag_9" )
      R_Coil( "中间变量值"."V_M_Q1.0" )
   END_RUNG
   // the same network as SCL:
   #_w1 := "S_循环水泵投入退出" AND "M_副井口#1泵手动启停" AND NOT "副井口循环泵手自状态反馈";
   #_w2 := #_w1 AND NOT "Tag_8";   // rising edge
   "Tag_8" := #_w1;
   IF #_w2 THEN "中间变量值"."V_M_Q1.0" := TRUE; END_IF;
   #_w3 := NOT #_w1 AND "Tag_9";   // falling edge
   "Tag_9" := #_w1;
   IF #_w3 THEN "中间变量值"."V_M_Q1.0" := FALSE; END_IF;
END_REGION

REGION Network 5: #2副井口输出中间变量
   RUNG wire#powerrail
      Contact( "S_循环水泵投入退出" )
      Contact( "M_副井口#2泵手动启停" )
      I_Contact( "副井口循环泵手自状态反馈" )
      wire#w1
      P_Trig( "Tag_10" )
      S_Coil( "中间变量值"."V_M_Q1.1" )
   END_RUNG
   RUNG wire#w1
      N_Trig( "Tag_11" )
      R_Coil( "中间变量值"."V_M_Q1.1" )
   END_RUNG
   // the same network as SCL:
   #_w1 := "S_循环水泵投入退出" AND "M_副井口#2泵手动启停" AND NOT "副井口循环泵手自状态反馈";
   #_w2 := #_w1 AND NOT "Tag_10";   // rising edge
   "Tag_10" := #_w1;
   IF #_w2 THEN "中间变量值"."V_M_Q1.1" := TRUE; END_IF;
   #_w3 := NOT #_w1 AND "Tag_11";   // falling edge
   "Tag_11" := #_w1;
   IF #_w3 THEN "中间变量值"."V_M_Q1.1" := FALSE; END_IF;
END_REGION

REGION Network 6: #3副井口输出中间变量
   RUNG wire#powerrail
      Contact( "S_循环水泵投入退出" )
      Contact( "M_副井口#3泵手动启停" )
      I_Contact( "副井口循环泵手自状态反馈" )
      wire#w1
      P_Trig( "Tag_12" )
      S_Coil( "中间变量值"."V_M_Q1.2" )
   END_RUNG
   RUNG wire#w1
      N_Trig( "Tag_13" )
      R_Coil( "中间变量值"."V_M_Q1.2" )
   END_RUNG
   // the same network as SCL:
   #_w1 := "S_循环水泵投入退出" AND "M_副井口#3泵手动启停" AND NOT "副井口循环泵手自状态反馈";
   #_w2 := #_w1 AND NOT "Tag_12";   // rising edge
   "Tag_12" := #_w1;
   IF #_w2 THEN "中间变量值"."V_M_Q1.2" := TRUE; END_IF;
   #_w3 := NOT #_w1 AND "Tag_13";   // falling edge
   "Tag_13" := #_w1;
   IF #_w3 THEN "中间变量值"."V_M_Q1.2" := FALSE; END_IF;
END_REGION

REGION Network 7: #1隔离泵控制输出中间变量
   RUNG wire#powerrail
      Contact( "S_循环水泵投入退出" )
      Contact( "M_隔离#1泵手动启停" )
      I_Contact( "#1隔离泵手自状态反馈" )
      wire#w1
      P_Trig( "Tag_14" )
      S_Coil( "中间变量值"."V_M_Q0.0" )
   END_RUNG
   RUNG wire#w1
      N_Trig( "Tag_15" )
      R_Coil( "中间变量值"."V_M_Q0.0" )
   END_RUNG
   // the same network as SCL:
   #_w1 := "S_循环水泵投入退出" AND "M_隔离#1泵手动启停" AND NOT "#1隔离泵手自状态反馈";
   #_w2 := #_w1 AND NOT "Tag_14";   // rising edge
   "Tag_14" := #_w1;
   IF #_w2 THEN "中间变量值"."V_M_Q0.0" := TRUE; END_IF;
   #_w3 := NOT #_w1 AND "Tag_15";   // falling edge
   "Tag_15" := #_w1;
   IF #_w3 THEN "中间变量值"."V_M_Q0.0" := FALSE; END_IF;
END_REGION

REGION Network 8: #2隔离泵控制输出中间变量
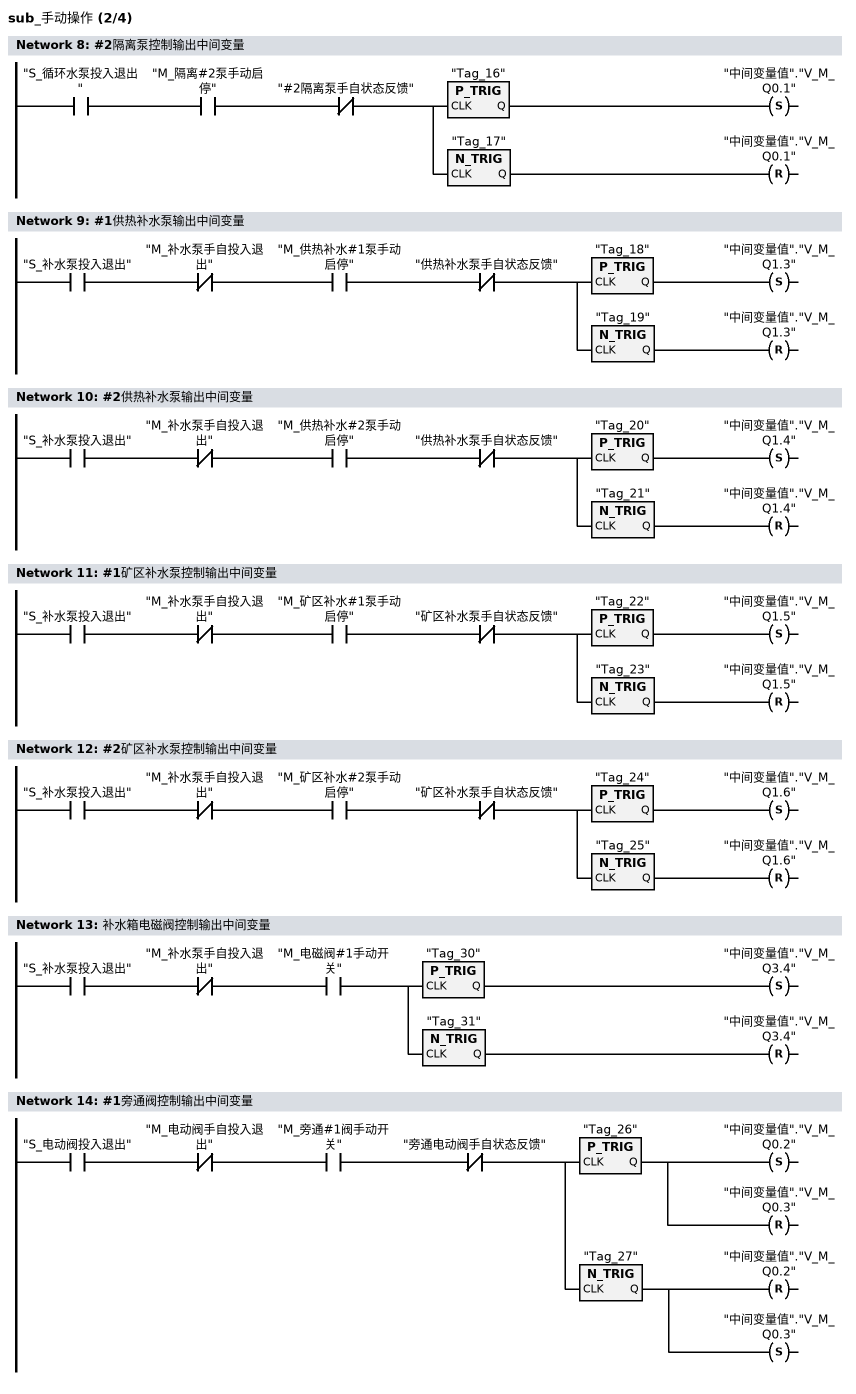
   RUNG wire#powerrail
      Contact( "S_循环水泵投入退出" )
      Contact( "M_隔离#2泵手动启停" )
      I_Contact( "#2隔离泵手自状态反馈" )
      wire#w1
      P_Trig( "Tag_16" )
      S_Coil( "中间变量值"."V_M_Q0.1" )
   END_RUNG
   RUNG wire#w1
      N_Trig( "Tag_17" )
      R_Coil( "中间变量值"."V_M_Q0.1" )
   END_RUNG
   // the same network as SCL:
   #_w1 := "S_循环水泵投入退出" AND "M_隔离#2泵手动启停" AND NOT "#2隔离泵手自状态反馈";
   #_w2 := #_w1 AND NOT "Tag_16";   // rising edge
   "Tag_16" := #_w1;
   IF #_w2 THEN "中间变量值"."V_M_Q0.1" := TRUE; END_IF;
   #_w3 := NOT #_w1 AND "Tag_17";   // falling edge
   "Tag_17" := #_w1;
   IF #_w3 THEN "中间变量值"."V_M_Q0.1" := FALSE; END_IF;
END_REGION

REGION Network 9: #1供热补水泵输出中间变量
   RUNG wire#powerrail
      Contact( "S_补水泵投入退出" )
      I_Contact( "M_补水泵手自投入退出" )
      Contact( "M_供热补水#1泵手动启停" )
      I_Contact( "供热补水泵手自状态反馈" )
      wire#w1
      P_Trig( "Tag_18" )
      S_Coil( "中间变量值"."V_M_Q1.3" )
   END_RUNG
   RUNG wire#w1
      N_Trig( "Tag_19" )
      R_Coil( "中间变量值"."V_M_Q1.3" )
   END_RUNG
   // the same network as SCL:
   #_w1 := "S_补水泵投入退出" AND NOT "M_补水泵手自投入退出" AND "M_供热补水#1泵手动启停" AND NOT "供热补水泵手自状态反馈";
   #_w2 := #_w1 AND NOT "Tag_18";   // rising edge
   "Tag_18" := #_w1;
   IF #_w2 THEN "中间变量值"."V_M_Q1.3" := TRUE; END_IF;
   #_w3 := NOT #_w1 AND "Tag_19";   // falling edge
   "Tag_19" := #_w1;
   IF #_w3 THEN "中间变量值"."V_M_Q1.3" := FALSE; END_IF;
END_REGION

REGION Network 10: #2供热补水泵输出中间变量
   RUNG wire#powerrail
      Contact( "S_补水泵投入退出" )
      I_Contact( "M_补水泵手自投入退出" )
      Contact( "M_供热补水#2泵手动启停" )
      I_Contact( "供热补水泵手自状态反馈" )
      wire#w1
      P_Trig( "Tag_20" )
      S_Coil( "中间变量值"."V_M_Q1.4" )
   END_RUNG
   RUNG wire#w1
      N_Trig( "Tag_21" )
      R_Coil( "中间变量值"."V_M_Q1.4" )
   END_RUNG
   // the same network as SCL:
   #_w1 := "S_补水泵投入退出" AND NOT "M_补水泵手自投入退出" AND "M_供热补水#2泵手动启停" AND NOT "供热补水泵手自状态反馈";
   #_w2 := #_w1 AND NOT "Tag_20";   // rising edge
   "Tag_20" := #_w1;
   IF #_w2 THEN "中间变量值"."V_M_Q1.4" := TRUE; END_IF;
   #_w3 := NOT #_w1 AND "Tag_21";   // falling edge
   "Tag_21" := #_w1;
   IF #_w3 THEN "中间变量值"."V_M_Q1.4" := FALSE; END_IF;
END_REGION

REGION Network 11: #1矿区补水泵控制输出中间变量
   RUNG wire#powerrail
      Contact( "S_补水泵投入退出" )
      I_Contact( "M_补水泵手自投入退出" )
      Contact( "M_矿区补水#1泵手动启停" )
      I_Contact( "矿区补水泵手自状态反馈" )
      wire#w1
      P_Trig( "Tag_22" )
      S_Coil( "中间变量值"."V_M_Q1.5" )
   END_RUNG
   RUNG wire#w1
      N_Trig( "Tag_23" )
      R_Coil( "中间变量值"."V_M_Q1.5" )
   END_RUNG
   // the same network as SCL:
   #_w1 := "S_补水泵投入退出" AND NOT "M_补水泵手自投入退出" AND "M_矿区补水#1泵手动启停" AND NOT "矿区补水泵手自状态反馈";
   #_w2 := #_w1 AND NOT "Tag_22";   // rising edge
   "Tag_22" := #_w1;
   IF #_w2 THEN "中间变量值"."V_M_Q1.5" := TRUE; END_IF;
   #_w3 := NOT #_w1 AND "Tag_23";   // falling edge
   "Tag_23" := #_w1;
   IF #_w3 THEN "中间变量值"."V_M_Q1.5" := FALSE; END_IF;
END_REGION

REGION Network 12: #2矿区补水泵控制输出中间变量
   RUNG wire#powerrail
      Contact( "S_补水泵投入退出" )
      I_Contact( "M_补水泵手自投入退出" )
      Contact( "M_矿区补水#2泵手动启停" )
      I_Contact( "矿区补水泵手自状态反馈" )
      wire#w1
      P_Trig( "Tag_24" )
      S_Coil( "中间变量值"."V_M_Q1.6" )
   END_RUNG
   RUNG wire#w1
      N_Trig( "Tag_25" )
      R_Coil( "中间变量值"."V_M_Q1.6" )
   END_RUNG
   // the same network as SCL:
   #_w1 := "S_补水泵投入退出" AND NOT "M_补水泵手自投入退出" AND "M_矿区补水#2泵手动启停" AND NOT "矿区补水泵手自状态反馈";
   #_w2 := #_w1 AND NOT "Tag_24";   // rising edge
   "Tag_24" := #_w1;
   IF #_w2 THEN "中间变量值"."V_M_Q1.6" := TRUE; END_IF;
   #_w3 := NOT #_w1 AND "Tag_25";   // falling edge
   "Tag_25" := #_w1;
   IF #_w3 THEN "中间变量值"."V_M_Q1.6" := FALSE; END_IF;
END_REGION

REGION Network 13: 补水箱电磁阀控制输出中间变量
   RUNG wire#powerrail
      Contact( "S_补水泵投入退出" )
      I_Contact( "M_补水泵手自投入退出" )
      Contact( "M_电磁阀#1手动开关" )
      wire#w1
      P_Trig( "Tag_30" )
      S_Coil( "中间变量值"."V_M_Q3.4" )
   END_RUNG
   RUNG wire#w1
      N_Trig( "Tag_31" )
      R_Coil( "中间变量值"."V_M_Q3.4" )
   END_RUNG
   // the same network as SCL:
   #_w1 := "S_补水泵投入退出" AND NOT "M_补水泵手自投入退出" AND "M_电磁阀#1手动开关";
   #_w2 := #_w1 AND NOT "Tag_30";   // rising edge
   "Tag_30" := #_w1;
   IF #_w2 THEN "中间变量值"."V_M_Q3.4" := TRUE; END_IF;
   #_w3 := NOT #_w1 AND "Tag_31";   // falling edge
   "Tag_31" := #_w1;
   IF #_w3 THEN "中间变量值"."V_M_Q3.4" := FALSE; END_IF;
END_REGION

REGION Network 14: #1旁通阀控制输出中间变量
   RUNG wire#powerrail
      Contact( "S_电动阀投入退出" )
      I_Contact( "M_电动阀手自投入退出" )
      Contact( "M_旁通#1阀手动开关" )
      I_Contact( "旁通电动阀手自状态反馈" )
      wire#w1
      P_Trig( "Tag_26" )
      wire#w2
      S_Coil( "中间变量值"."V_M_Q0.2" )
   END_RUNG
   RUNG wire#w2
      R_Coil( "中间变量值"."V_M_Q0.3" )
   END_RUNG
   RUNG wire#w1
      N_Trig( "Tag_27" )
      wire#w3
      R_Coil( "中间变量值"."V_M_Q0.2" )
   END_RUNG
   RUNG wire#w3
      S_Coil( "中间变量值"."V_M_Q0.3" )
   END_RUNG
   // the same network as SCL:
   #_w1 := "S_电动阀投入退出" AND NOT "M_电动阀手自投入退出" AND "M_旁通#1阀手动开关" AND NOT "旁通电动阀手自状态反馈";
   #_w2 := #_w1 AND NOT "Tag_26";   // rising edge
   "Tag_26" := #_w1;
   IF #_w2 THEN
       "中间变量值"."V_M_Q0.2" := TRUE;
       "中间变量值"."V_M_Q0.3" := FALSE;
   END_IF;
   #_w3 := NOT #_w1 AND "Tag_27";   // falling edge
   "Tag_27" := #_w1;
   IF #_w3 THEN
       "中间变量值"."V_M_Q0.2" := FALSE;
       "中间变量值"."V_M_Q0.3" := TRUE;
   END_IF;
END_REGION

REGION Network 15: #2旁通阀输出中间变量
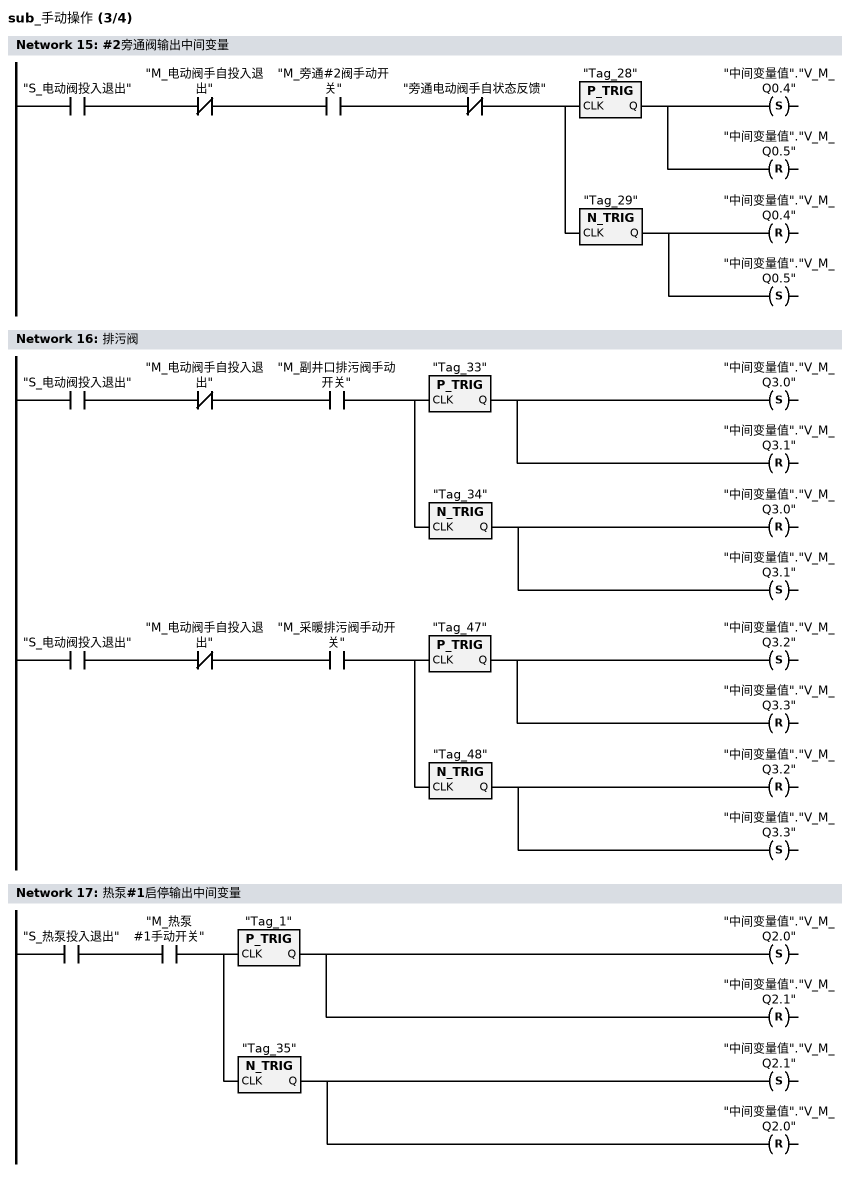
   RUNG wire#powerrail
      Contact( "S_电动阀投入退出" )
      I_Contact( "M_电动阀手自投入退出" )
      Contact( "M_旁通#2阀手动开关" )
      I_Contact( "旁通电动阀手自状态反馈" )
      wire#w1
      P_Trig( "Tag_28" )
      wire#w2
      S_Coil( "中间变量值"."V_M_Q0.4" )
   END_RUNG
   RUNG wire#w2
      R_Coil( "中间变量值"."V_M_Q0.5" )
   END_RUNG
   RUNG wire#w1
      N_Trig( "Tag_29" )
      wire#w3
      R_Coil( "中间变量值"."V_M_Q0.4" )
   END_RUNG
   RUNG wire#w3
      S_Coil( "中间变量值"."V_M_Q0.5" )
   END_RUNG
   // the same network as SCL:
   #_w1 := "S_电动阀投入退出" AND NOT "M_电动阀手自投入退出" AND "M_旁通#2阀手动开关" AND NOT "旁通电动阀手自状态反馈";
   #_w2 := #_w1 AND NOT "Tag_28";   // rising edge
   "Tag_28" := #_w1;
   IF #_w2 THEN
       "中间变量值"."V_M_Q0.4" := TRUE;
       "中间变量值"."V_M_Q0.5" := FALSE;
   END_IF;
   #_w3 := NOT #_w1 AND "Tag_29";   // falling edge
   "Tag_29" := #_w1;
   IF #_w3 THEN
       "中间变量值"."V_M_Q0.4" := FALSE;
       "中间变量值"."V_M_Q0.5" := TRUE;
   END_IF;
END_REGION

REGION Network 16: 排污阀
   RUNG wire#powerrail
      Contact( "S_电动阀投入退出" )
      I_Contact( "M_电动阀手自投入退出" )
      Contact( "M_副井口排污阀手动开关" )
      wire#w1
      P_Trig( "Tag_33" )
      wire#w2
      S_Coil( "中间变量值"."V_M_Q3.0" )
   END_RUNG
   RUNG wire#w2
      R_Coil( "中间变量值"."V_M_Q3.1" )
   END_RUNG
   RUNG wire#w1
      N_Trig( "Tag_34" )
      wire#w3
      R_Coil( "中间变量值"."V_M_Q3.0" )
   END_RUNG
   RUNG wire#w3
      S_Coil( "中间变量值"."V_M_Q3.1" )
   END_RUNG
   RUNG wire#powerrail
      Contact( "S_电动阀投入退出" )
      I_Contact( "M_电动阀手自投入退出" )
      Contact( "M_采暖排污阀手动开关" )
      wire#w4
      P_Trig( "Tag_47" )
      wire#w5
      S_Coil( "中间变量值"."V_M_Q3.2" )
   END_RUNG
   RUNG wire#w5
      R_Coil( "中间变量值"."V_M_Q3.3" )
   END_RUNG
   RUNG wire#w4
      N_Trig( "Tag_48" )
      wire#w6
      R_Coil( "中间变量值"."V_M_Q3.2" )
   END_RUNG
   RUNG wire#w6
      S_Coil( "中间变量值"."V_M_Q3.3" )
   END_RUNG
   // the same network as SCL:
   #_w1 := "S_电动阀投入退出" AND NOT "M_电动阀手自投入退出" AND "M_副井口排污阀手动开关";
   #_w2 := #_w1 AND NOT "Tag_33";   // rising edge
   "Tag_33" := #_w1;
   IF #_w2 THEN
       "中间变量值"."V_M_Q3.0" := TRUE;
       "中间变量值"."V_M_Q3.1" := FALSE;
   END_IF;
   #_w3 := NOT #_w1 AND "Tag_34";   // falling edge
   "Tag_34" := #_w1;
   IF #_w3 THEN
       "中间变量值"."V_M_Q3.0" := FALSE;
       "中间变量值"."V_M_Q3.1" := TRUE;
   END_IF;
   #_w4 := "S_电动阀投入退出" AND NOT "M_电动阀手自投入退出" AND "M_采暖排污阀手动开关";
   #_w5 := #_w4 AND NOT "Tag_47";   // rising edge
   "Tag_47" := #_w4;
   IF #_w5 THEN
       "中间变量值"."V_M_Q3.2" := TRUE;
       "中间变量值"."V_M_Q3.3" := FALSE;
   END_IF;
   #_w6 := NOT #_w4 AND "Tag_48";   // falling edge
   "Tag_48" := #_w4;
   IF #_w6 THEN
       "中间变量值"."V_M_Q3.2" := FALSE;
       "中间变量值"."V_M_Q3.3" := TRUE;
   END_IF;
END_REGION

REGION Network 17: 热泵#1启停输出中间变量
   RUNG wire#powerrail
      Contact( "S_热泵投入退出" )
      Contact( "M_热泵 #1手动开关" )
      wire#w1
      P_Trig( "Tag_1" )
      wire#w2
      S_Coil( "中间变量值"."V_M_Q2.0" )
   END_RUNG
   RUNG wire#w2
      R_Coil( "中间变量值"."V_M_Q2.1" )
   END_RUNG
   RUNG wire#w1
      N_Trig( "Tag_35" )
      wire#w3
      S_Coil( "中间变量值"."V_M_Q2.1" )
   END_RUNG
   RUNG wire#w3
      R_Coil( "中间变量值"."V_M_Q2.0" )
   END_RUNG
   // the same network as SCL:
   #_w1 := "S_热泵投入退出" AND "M_热泵 #1手动开关";
   #_w2 := #_w1 AND NOT "Tag_1";   // rising edge
   "Tag_1" := #_w1;
   IF #_w2 THEN
       "中间变量值"."V_M_Q2.0" := TRUE;
       "中间变量值"."V_M_Q2.1" := FALSE;
   END_IF;
   #_w3 := NOT #_w1 AND "Tag_35";   // falling edge
   "Tag_35" := #_w1;
   IF #_w3 THEN
       "中间变量值"."V_M_Q2.1" := TRUE;
       "中间变量值"."V_M_Q2.0" := FALSE;
   END_IF;
END_REGION

REGION Network 18: 热泵#2启停输出中间变量
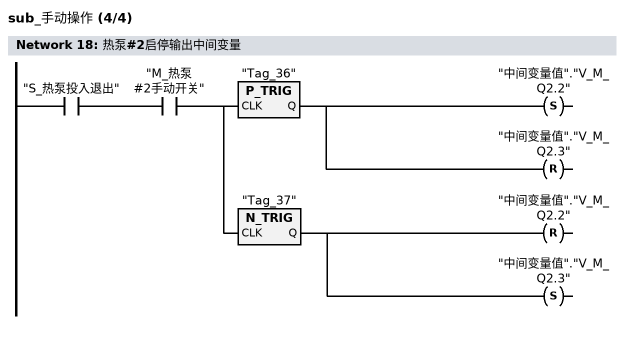
   RUNG wire#powerrail
      Contact( "S_热泵投入退出" )
      Contact( "M_热泵 #2手动开关" )
      wire#w1
      P_Trig( "Tag_36" )
      wire#w2
      S_Coil( "中间变量值"."V_M_Q2.2" )
   END_RUNG
   RUNG wire#w2
      R_Coil( "中间变量值"."V_M_Q2.3" )
   END_RUNG
   RUNG wire#w1
      N_Trig( "Tag_37" )
      wire#w3
      R_Coil( "中间变量值"."V_M_Q2.2" )
   END_RUNG
   RUNG wire#w3
      S_Coil( "中间变量值"."V_M_Q2.3" )
   END_RUNG
   // the same network as SCL:
   #_w1 := "S_热泵投入退出" AND "M_热泵 #2手动开关";
   #_w2 := #_w1 AND NOT "Tag_36";   // rising edge
   "Tag_36" := #_w1;
   IF #_w2 THEN
       "中间变量值"."V_M_Q2.2" := TRUE;
       "中间变量值"."V_M_Q2.3" := FALSE;
   END_IF;
   #_w3 := NOT #_w1 AND "Tag_37";   // falling edge
   "Tag_37" := #_w1;
   IF #_w3 THEN
       "中间变量值"."V_M_Q2.2" := FALSE;
       "中间变量值"."V_M_Q2.3" := TRUE;
   END_IF;
END_REGION
END_ORGANIZATION_BLOCK